FUNCTION_BLOCK subMat
VAR_INPUT
	a:REFERENCE TO Array2DStaticMatrix;
	b:REFERENCE TO Array2DStaticMatrix;
	c:REFERENCE TO Array2DStaticMatrix;
	m,n:INT;
END_VAR
VAR_OUTPUT
END_VAR
VAR
	i,j:int;
END_VAR

 

    FOR i:=0 TO m DO
        FOR j:=0TO n DO
            c[i*n+j] := a[i*n+j]-b[i*n+j];
			END_FOR
			END_FOR

END_FUNCTION_BLOCK

(* stored: Version 1.1.0.1, ProductVersion 3.1.4024.12
   POU subMat: Id {29b4e301-1fb7-446e-b08d-551b8a88f591}, SpecialFunc None *)
